Yaskawa INFORM job: SIDE-A-CLAMP.JBI

/JOB
//NAME SIDE-A-CLAMP
///FOLDERNAME CLAMPUNCLAMP
//POS
///NPOS 0,0,0,0,0,0
//INST
///DATE 2021/10/04 12:16
///ATTR SC,RW
NOP
'********************************
'CLOSE CLAMP
'SIDE-A ARW CELL#2
'********************************
SET B099 0
'**CLOSE CLAMP**
DOUT OT#(137) OFF
DOUT OT#(138) ON
WAIT IN#(141)=ON T=3.00
JUMP *QUIT IF IN#(141)=OFF
'**CLAMPING COMPLETE**
SET B099 1
*QUIT
END
